ABB RobotStudio station: Tp2_20201216-052747.rsstn

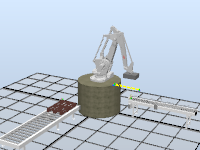
Station Tp2 (saved by RobotStudio 20.2.9116.0)
Controller Controlador1
  mechanical unit ROB_1: IRB660_180_315__01_2, 6 joints, base frame (0, 0, 1500) mm
Layout (positions relative to the parent item):
  - transporteCajas [part, from Equipment\Conveyor Guide 400.rslib] at (0, 1500, 0) mm, rotated rx 0 ry 0 rz 90 deg
  - Euro Pallet [graphiccomponentgroup, from Equipment\Euro Pallet.rslib] at (1000, -1425, 435) mm
    - Body 1 [part, from Equipment\Euro Pallet.rslib]
  - transportePallets [part, from Equipment\Conveyor 950 4000 h2.rslib] at (1000, -1500, 0) mm
  - IRB660_180_315__01_2 [mechanism, from Robots\IRB660_180_315__01.rslib] at (0, 0, 1500) mm; joint values [1.7033, 0.3901, 1.218, 1.7033] (rad or m)
  - ventosa_tool [mechanism] at (-200, 1500, 1970) mm, rotated rx 180 ry 0 rz 180 deg
      TCP ventosa_tool at (0, 0, 200) mm
      links: ventosa
  - fuenteBloques [smart component] at (-200, 1500, 770) mm
      signals: DI agarrar, DO cajaLista
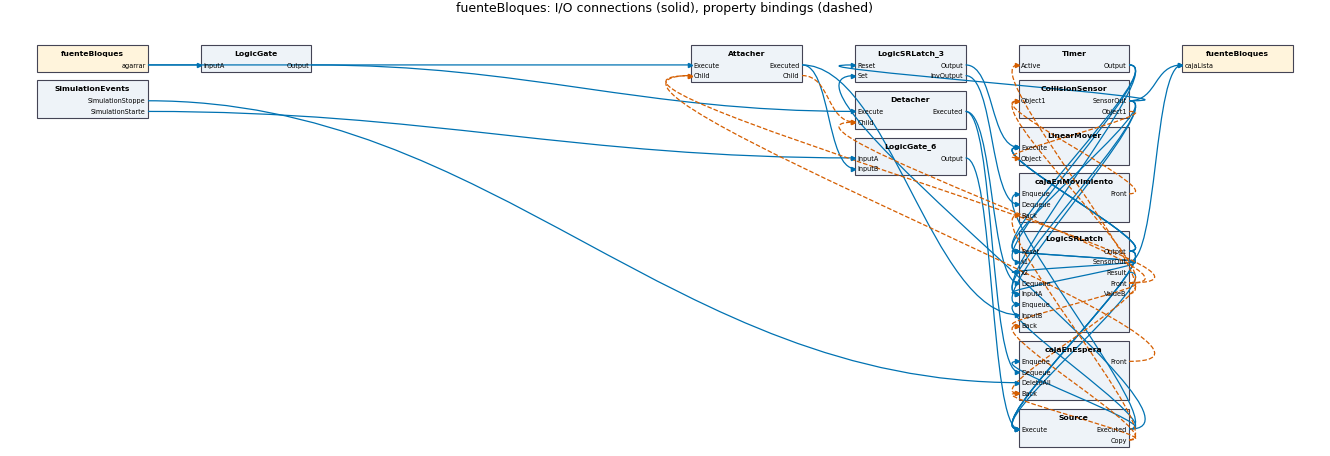
      connections:
        LogicSRLatch.Output -> LinearMover.Execute
        PlaneSensor.SensorOut -> LogicSRLatch.Reset
        Timer.Output -> LogicExpression.x1
        PlaneSensor.SensorOut -> LogicExpression.x2
        LogicExpression.Result -> Source.Execute
        PlaneSensor.SensorOut -> fuenteBloques.cajaLista
        LogicGate.Output -> Detacher.Execute
        fuenteBloques.agarrar -> LogicGate.InputA
        Detacher.Executed -> cajasEnEspera.Dequeue
        PlaneSensor.SensorOut -> LogicGate_2.InputA
        LogicSRLatch.Output -> LinearMover.Execute
        PlaneSensor.SensorOut -> LogicSRLatch.Reset
        CollisionSensor.SensorOut -> LogicSRLatch.Reset
        CollisionSensor.SensorOut -> fuenteBloques.cajaLista
        LogicGate_3.Output -> LinearMover.Execute
        CollisionSensor.SensorOut -> LogicGate_3.InputA
        Source.Executed -> cajasMoviendose.Enqueue
        CollisionSensor.SensorOut -> cajasEnEspera.Enqueue
        fuenteBloques.agarrar -> Attacher.Execute
        Source.Executed -> cajaEnEspera.Enqueue
        Detacher.Executed -> cajaEnEspera.Dequeue
        LogicGate_4.Output -> Source.Execute
        LogicSRLatch_2.Output -> Source.Execute
        Timer.Output -> LogicSRLatch_2.Reset
        LogicGate_5.Output -> Source.Execute
        Timer.Output -> LogicGate_5.InputA
        Attacher.Executed -> LogicGate_5.InputB
        LogicSRLatch_3.Output -> LinearMover.Execute
        CollisionSensor.SensorOut -> LogicSRLatch_3.Reset
        Source.Executed -> LogicSRLatch_3.Set
        Source.Executed -> cajaEnMovimiento.Enqueue
        LogicSRLatch_3.InvOutput -> cajaEnMovimiento.Dequeue
        SimulationEvents.SimulationStopped -> cajaEnEspera.DeleteAll
        SimulationEvents.SimulationStarted -> LogicGate_6.InputA
        LogicGate_6.Output -> Source.Execute
        Attacher.Executed -> LogicGate_6.InputB
        cajasEnEspera.Front => Attacher.Child
        cajasEnEspera.Front => Detacher.Child
        CollisionSensor.Object1 => LinearMover.Object
        Source.Copy => cajasMoviendose.Back
        cajasMoviendose.Front => CollisionSensor.Object1
        cajasMoviendose.Front => cajasEnEspera.Back
        Attacher.Child => Detacher.Child
        cajaEnEspera.Front => Attacher.Child
        cajasMoviendose.Front => cajaEnEspera.Back
        Source.Copy => cajaEnEspera.Back
        Source.Copy => cajaEnMovimiento.Back
        cajaEnMovimiento.Front => CollisionSensor.Object1
        Comparer.ValueB => Timer.Active
    - Source [smart component, from Components\Source.rslib]
        properties: Source=caja; Copy=(none); Parent=(none); Position=[0 2.5 0]; Orientation=[0 0 0]; Transient=true; PhysicsBehavior=0
    - Timer [smart component, from Components\Timer.rslib]
        properties: StartTime=0; Interval=5; Repeat=true; CurrentTime=174.84
    - LinearMover [smart component, from Components\LinearMover.rslib]
        properties: Object=(none); Direction=[0 1 0]; Speed=-0.2; Reference=Object; ReferenceObject=fuenteBloques
    - caja [part]
    - Attacher [smart component, from Components\Attacher.rslib]
        properties: Parent=ventosa_tool; Flange=0; Child=(none); Mount=false; Offset=[0 0 0]; Orientation=[0 0 0]
    - Detacher [smart component, from Components\Detacher.rslib]
        properties: Child=(none); KeepPosition=true
    - StopSimulation [smart component, from Components\StopSimulation.rslib]
    - StopSimulation_2 [smart component, from Components\StopSimulation.rslib]
    - LogicGate [smart component, from Components\LogicGate.rslib]
        properties: Operator=NOT; Delay=0
    - CollisionSensor [smart component, from Components\CollisionSensor.rslib]
        properties: Object1=(none); Object2=sensorCaja; NearMiss=0; Part1=(none); Part2=sensorCaja; CollisionType=2
    - sensorCaja [part] at (-100, 1, 0) mm, rotated rx 90 ry 0 rz 0 deg
    - cajaEnEspera [smart component, from Components\Queue.rslib]
        properties: Back=(none); Front=(none); Queue=; NumberOfObjects=0
    - LogicSRLatch_3 [smart component, from Components\LogicSRLatch.rslib]
    - cajaEnMovimiento [smart component, from Components\Queue.rslib]
        properties: Back=(none); Front=(none); Queue={1c2bc98a-7e79-4a64-8c08-18c22f355a99};{e1edf675-8202-4f71-9da3-817a982703fd};{ffd251ec-a3cf-41ee-8966-fdd0fbeca7f4};{f1d19616-4be7-4e79-a789-1261585d2031};{093a5ca0-ccf5-4320-a6b7-bb8c054aae36};{df3f017b-7df1-41a5-aac6-cc923bf41019};{7c2eaaf3-8dec-4732-9310-3e721976978d};{45dc22b4-1054-4488-b7ca-ac52e89d740b};{5a8c4baf-114b-4097-b143-104adfb42322};{6b3b95f4-b342-4a81-929e-5c9f996cfed1};{ece14d91-df30-41b2-b85e-dd972d5a8e39};{c7e8cb03-728e-4264-a3ea-bfc9f1c7ddce};{ab919f7f-0554-446b-a56d-53fbfc5d8ce7};{a30dad3d-a8f1-47db-80a1-64ec5784e0b4};{19c0da7d-87c3-4e24-a10a-9007f1d8b843};{d8cc487c-9e99-461b-bbdf-f4737f623ea7};{8687cdd6-b602-47a9-b251-d4b979f610a2};{4c41ed51-1b61-46b0-9096-6d1030f11c3b};{a1fc6fb9-ef4e-4696-8b79-4e61b0871820};{e91b887a-1e53-4284-a6ce-b383082e36d3};{4c35c9c7-266f-4545-9d66-60066f554cc2};{341bfa75-53ee-4b2b-a5d1-76565c96955c};{ea93a2cb-1666-4ed6-a9de-bbf598504c3d};{81eee15b-9bd5-422a-a729-479eb919e521};{659a2bd0-144c-468a-bc5f-a7357c1e4eaa};{20785ed1-5c16-412f-8c62-e2f0240c2008}; NumberOfObjects=0
    - SimulationEvents [smart component, from Components\SimulationEvents.rslib]
    - LogicGate_6 [smart component, from Components\LogicGate.rslib]
        properties: Operator=OR; Delay=0
  - Pedestal [part]
Attachment: Euro Pallet is attached to transportePallets
Attachment: ventosa_tool is attached to IRB660_180_315__01_2 / Link6
Attachment: pistaCajas is attached to transporteCajas
Attachment: pistaPallets is attached to transportePallets
Station logic (signal -> signal, property => property):
  Controlador1.do_pick -> fuenteBloques.agarrar
  fuenteBloques.cajaLista -> Controlador1.cajaLista
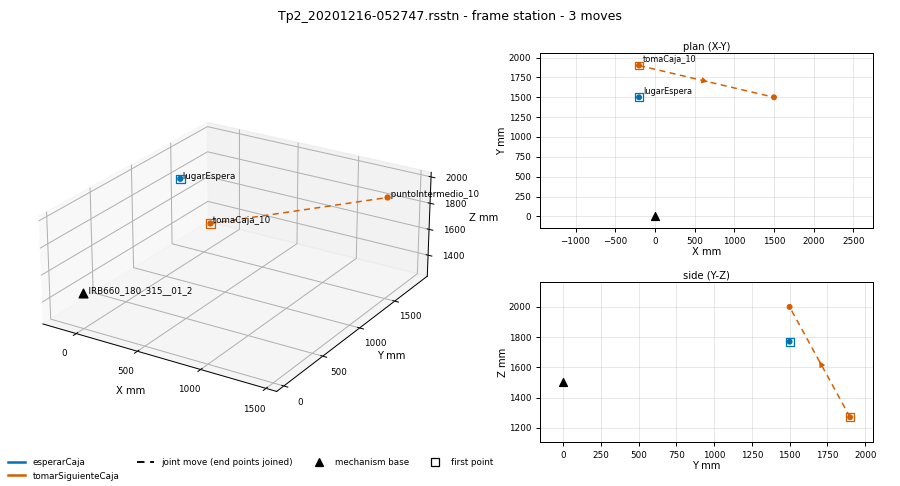
[picture p0: tool path of Tp2_20201216-052747.rsstn in frame station, 3 of 3 moves have a stored position in this frame; points joined in program order, loops and branches not executed]
Targets, tools, work objects and paths stored in the station, written as RAPID:
! task T_ROB1
MODULE Module1
  PERS tooldata ventosa_tool:=[TRUE,[[0,0,200],[1,0,0,0]],[1,[0,0,1],[1,0,0,0],0,0,0]];
  PERS wobjdata pistaCajas:=[FALSE,TRUE,"",[[-200,1500,770],[0,0,1,0]],[[0,0,0],[1,0,0,0]]];
  PERS wobjdata pistaPallets:=[FALSE,TRUE,"",[[1000,-1425,579],[0,0,1,0]],[[0,0,0],[1,0,0,0]]];
  CONST robtarget lugarEspera:=[[0,0,-1000],[1,0,0,0],[0,0,0,0],[9E+09,9E+09,9E+09,9E+09,9E+09,9E+09]];
  CONST robtarget tomaCaja_10:=[[0,400,-500],[1,0,0,0],[0,0,0,0],[9E+09,9E+09,9E+09,9E+09,9E+09,9E+09]];
  CONST robtarget superficiePallet_10:=[[0,0,0],[1,0,0,0],[0,0,0,0],[9E+09,9E+09,9E+09,9E+09,9E+09,9E+09]];
  CONST robtarget puntoIntermedio_10:=[[1500,1500,2000],[0,0,1,0],[0,0,0,0],[9E+09,9E+09,9E+09,9E+09,9E+09,9E+09]];
  PROC main()
    SetDO do_pick,0;
    esperarCaja;
    tomarSiguienteCaja;
    esperarCaja;
  ENDPROC
  PROC esperarCaja()
    MoveJ lugarEspera,v1000,fine,ventosa_tool\WObj:=pistaCajas;
    WaitDI cajaLista,1;
  ENDPROC
  PROC tomarSiguienteCaja()
    MoveJ tomaCaja_10,v1000,fine,ventosa_tool\WObj:=pistaCajas;
    SetDO do_pick,1;
    WaitTime 0.2;
    MoveJ puntoIntermedio_10,v1000,z100,ventosa_tool\WObj:=wobj0;
  ENDPROC
ENDMODULE

